INTERFACE I_Mediator

METHOD notify : BOOL
VAR_INPUT
	// Colleague sending the notification
	sender : I_Colleague;
	// Some event the collegue is attempting
	event	  : STRING;
END_VAR
END_METHOD

END_INTERFACE

(* stored: Version 1.1.0.1, ProductVersion 3.1.4024.12
   Itf I_Mediator: Id {bdafaeae-011d-481a-9d42-ca799f98d128}
   Method notify: Id {22fcc692-7d51-4d94-b380-7ccd6f446c31} *)
